PROGRAM MAIN
VAR
END_VAR

;

END_PROGRAM

(* stored: Version 1.1.0.1, ProductVersion 3.1.4024.6
   POU MAIN: Id {7a0c6b10-31d2-445f-aa5f-902e41ceca90}, SpecialFunc None *)
